TYPE MonitoredValue :
STRUCT
	rawValue          : INT;
	rawValueMin       : INT;
	rawValueMax       : INT;
	scaledValue       : REAL;
	scaledValueMin    : REAL;
	scaledValueMax    : REAL;
	units             : STRING(10);
	lowerWarningValue : REAL;
	upperWarningValue : REAL; 
	dbName            : STRING(50);
END_STRUCT
END_TYPE

(* stored: Version 1.1.0.1, ProductVersion 3.1.4024.12
   DUT MonitoredValue: Id {566712ed-280a-4222-a0fc-b368ed44a062} *)
